{attribute 'GeneratedUsingTerminal: EL6731--0000'}
{attribute addProperty BoxType "EL6731--0000"}
{attribute addProperty Id "InfoDataAT %I*InfoData_41C547A32"}
{attribute addProperty CRC "3204926373"}
{attribute addProperty Size "2"}
TYPE EL6731_BF074BA5 EXTENDS EtcSlaveTerminalBase_947E5A46 :
STRUCT
	{attribute addProperty Name "InfoData"}
	InfoData : InfoData_41C547A3;
END_STRUCT
END_TYPE

(* stored: Version 1.2.0.0, ProductVersion 3.1.4024.9
   DUT EL6731_BF074BA5: Id {d518606b-74a4-4f1c-8fa4-099d8bb08c31} *)
